INTERFACE I_XtsMover

PROPERTY Acceleration : mc_lreal
GET
END_GET
SET
END_SET
END_PROPERTY

METHOD ActivateTrack : HRESULT
VAR_INPUT
	Track : INT;
END_VAR
END_METHOD

METHOD ActivateZeroReferenceSystem : HRESULT
END_METHOD

PROPERTY ActualForce : LREAL
GET
END_GET
END_PROPERTY

PROPERTY ActualPosition : LREAL
GET
END_GET
END_PROPERTY

PROPERTY ActualTrackPosition : LREAL
GET
END_GET
END_PROPERTY

PROPERTY ActualVelocity : LREAL
GET
END_GET
END_PROPERTY

PROPERTY AxisRef : Reference to Axis_ref
GET
END_GET
END_PROPERTY

PROPERTY Deceleration : mc_lreal
GET
END_GET
SET
END_SET
END_PROPERTY

METHOD DisableMover : HRESULT
VAR_INPUT
END_VAR
END_METHOD

METHOD EnableMover : HRESULT
VAR_INPUT
END_VAR
END_METHOD

PROPERTY ErrorID : UDINT
GET
END_GET
END_PROPERTY

PROPERTY Gap : MC_LREAL
GET
END_GET
SET
END_SET
END_PROPERTY

METHOD GetActiveTrackLength : LREAL
VAR_INPUT
END_VAR
END_METHOD

METHOD GetMoverCtrlOTCID : XtsMoverControllerOTCID
VAR_INPUT
END_VAR
END_METHOD

METHOD HaltAxis : HRESULT
VAR_INPUT
END_VAR
END_METHOD

PROPERTY HasError : BOOL
GET
END_GET
END_PROPERTY

PROPERTY PUBLIC IdentInGroup : IDENT_IN_GROUP_REF
GET
END_GET
END_PROPERTY

PROPERTY IsActive : BOOL
GET
END_GET
END_PROPERTY

PROPERTY IsAMover1 : BOOL
GET
END_GET
END_PROPERTY

PROPERTY IsAvoidingCollision : BOOL
GET
END_GET
END_PROPERTY

PROPERTY IsDetected : BOOL
GET
END_GET
END_PROPERTY

PROPERTY IsEnabled : BOOL
GET
END_GET
END_PROPERTY

PROPERTY IsStationary : BOOL
GET
END_GET
END_PROPERTY

PROPERTY Jerk : mc_lreal
GET
END_GET
SET
END_SET
END_PROPERTY

PROPERTY PUBLIC MoversActiveTrack : INT
GET
END_GET
END_PROPERTY

PROPERTY PUBLIC MoverXtsIoEnvInterface : I_TcIoXtsXpuMover
GET
END_GET
SET
END_SET
END_PROPERTY

METHOD MoveTo : HRESULT
VAR_INPUT
	RequiredPosition : MC_LREAL;
	MoveVelocity : MC_LREAL;
	NonModuloMove : BOOL;
END_VAR
END_METHOD

PROPERTY MyCAGroup : I_CollisionGroup
GET
END_GET
SET
END_SET
END_PROPERTY

PROPERTY PositiveDirectionOnly : BOOL
GET
END_GET
SET
END_SET
END_PROPERTY

METHOD RegisterTracks : HRESULT
VAR_INPUT
	Track : I_XtsTrack;
END_VAR
END_METHOD

METHOD Reset : HRESULT
VAR_INPUT
END_VAR
END_METHOD

METHOD SetForceCouple : HRESULT
VAR_INPUT
	XtsMoverCtrlOTCID : Tc3_XTS_Utility.XtsMoverControllerOTCID;
END_VAR
END_METHOD

METHOD SetMoverActiveTrack : HRESULT
VAR_INPUT
	Track : INT;
END_VAR
END_METHOD

METHOD SetParameterSet : HRESULT
VAR_INPUT
	ParameterSet : OTCID;
END_VAR
END_METHOD

METHOD SetSimDetectionPartAndPosition : BOOL
VAR_INPUT
	Part : OTCID;
	Position : LREAL;
END_VAR
END_METHOD

METHOD TriggerMoverArrive : HRESULT
VAR_INPUT
END_VAR
END_METHOD

METHOD TriggerMoverLeave : HRESULT
VAR_INPUT
END_VAR
END_METHOD

END_INTERFACE

(* stored: Version 1.1.0.1
   Itf I_XtsMover: Id {3dcfc709-5ede-408c-bb46-9ff1ab7ba3a2}
   Folder Administration: Id {4954b02a-5467-474b-b4cc-9e953c27295d}
   Folder Commands: Id {106fb726-2896-4a76-8d42-ca08d03a1871}
   Folder Dynamics: Id {f06c35fd-2445-4fb9-97b8-caf92ac08b38}
   Folder Status: Id {6f079834-b92a-4de6-abe6-7b90d541a1af}
   Property Acceleration: Id {968dd06c-5bd7-474e-8a7d-3c6c7a848d78}
   Get Get: Id {ad3ccb1b-ebe0-4c79-851d-54fe9678941a}
   Set Set: Id {ad0cd55c-ffe5-41e5-89e5-44c936340625}
   Method ActivateTrack: Id {ba6e327e-25a9-4189-a1a0-64429eeca8b6}
   Method ActivateZeroReferenceSystem: Id {ab0eeb60-9673-46f5-be7f-8e50f8587ea1}
   Property ActualForce: Id {00e4b1c4-c6de-437f-8c1d-7314c009badc}
   Get Get: Id {ae9db5cd-10af-4e87-b4a2-e547ec5c553c}
   Property ActualPosition: Id {28cc63bc-e59d-4da9-a15c-a10a220bddfe}
   Get Get: Id {9cdf084e-f593-4336-8f01-56fe49195bb3}
   Property ActualTrackPosition: Id {e9f1d418-aa47-422b-9743-bf025f0e00db}
   Get Get: Id {5f8e75a9-0ebf-4529-928e-062c555b8cba}
   Property ActualVelocity: Id {4743bebc-3e65-4ae0-ae76-394e50299433}
   Get Get: Id {c9377cd8-6623-42ce-ab9c-71b02227228b}
   Property AxisRef: Id {b9459322-2642-4758-9d1a-f140abbed4b3}
   Get Get: Id {fca9e840-ce68-48f6-aaf7-b30da4df166b}
   Property Deceleration: Id {925224a3-633f-4afb-a6bb-5e2282bf0166}
   Get Get: Id {ee77943b-5dd1-4851-bfac-c1f6c08f427a}
   Set Set: Id {cf0b19b4-9657-4139-bc2e-afb49fbc4d88}
   Method DisableMover: Id {ab15092e-3fa3-489a-9dc6-5a5b357cf3f5}
   Method EnableMover: Id {12e4840c-ab85-431d-8aa9-ce712b4847e4}
   Property ErrorID: Id {b04c2e44-101b-40a1-bb51-ba2468016913}
   Get Get: Id {4e6c86e3-a90a-4b81-8f9a-ac29a4c9cc2b}
   Property Gap: Id {fb9a5121-dbab-42c7-b05b-e0e4367182c8}
   Get Get: Id {0b18224e-8e16-4474-96e3-0906bc0c9a81}
   Set Set: Id {2dea6ad0-842c-4a1e-91cb-fd845bae918b}
   Method GetActiveTrackLength: Id {5c2216e1-42a4-4136-9c70-0f82d23b2aef}
   Method GetMoverCtrlOTCID: Id {863e8ade-d7f2-439e-8b15-5f1837c580a0}
   Method HaltAxis: Id {881642ff-213b-4030-944f-bd624c008c64}
   Property HasError: Id {90e38746-64a9-412e-b69f-e80f2d788cc6}
   Get Get: Id {5d936f5b-33ae-4901-8b9f-50eb63a5b11c}
   Property IdentInGroup: Id {892b953d-abf1-49a8-bf89-421385c1791d}
   Get Get: Id {b023befb-8f40-468b-ada4-daaf368f7d24}
   Property IsActive: Id {43095e03-0781-4c14-aea8-4bb8d9b5c9a9}
   Get Get: Id {5c30f132-658c-45bd-986b-b41d82b1ab82}
   Property IsAMover1: Id {2bbcc45a-af5d-48fd-a64e-6509262e5e53}
   Get Get: Id {35cbc1b6-e96d-405e-9119-f59168018c94}
   Property IsAvoidingCollision: Id {5943782e-d40c-4ea0-9ddf-8fe8e953cf52}
   Get Get: Id {a0bd6fb0-24f5-415f-851e-6efe2481bd7c}
   Property IsDetected: Id {93c73707-2737-4a0d-b791-8a8c892ba285}
   Get Get: Id {5a7d46d0-a531-4a2d-8d8f-a2055343f49b}
   Property IsEnabled: Id {1dc642f1-9317-4da4-80d2-54b08fffd57c}
   Get Get: Id {0b3bdbce-a4ec-4a95-bc52-fef9dadad358}
   Property IsStationary: Id {08154e2f-b533-419e-9633-c8866a41fb11}
   Get Get: Id {4afa1b23-4ee3-47ce-9d91-4217690a4938}
   Property Jerk: Id {8063437d-ace9-4769-bdaf-bbbe2e6cdcb8}
   Get Get: Id {7a71a7bc-503a-407e-bd5c-807dc27f8a07}
   Set Set: Id {943274ff-ff90-4228-a079-22863adf0d58}
   Property MoversActiveTrack: Id {f033ba71-1699-4f66-8762-38178a524724}
   Get Get: Id {ab30b8a7-22d3-4a5c-a941-ce17b5400c54}
   Property MoverXtsIoEnvInterface: Id {192fc175-f0e7-4171-9425-47deb3799f9d}
   Get Get: Id {e7a8a250-ae9b-4ad7-bf97-7690d04cb985}
   Set Set: Id {f163ce07-1471-4036-baf2-4d783308d9bd}
   Method MoveTo: Id {ff1a94f0-d91e-4f1f-8540-ce9d25779d5e}
   Property MyCAGroup: Id {7bdbd73e-c8bd-4342-9139-b02fb8b34afa}
   Get Get: Id {02d1886c-e164-4472-af91-ae6725f23e23}
   Set Set: Id {0add7ecc-1e34-4c45-86ea-05d00a10668e}
   Property PositiveDirectionOnly: Id {ed0ab13d-fd6f-4b8b-a5b2-30d977b85665}
   Get Get: Id {ca7928e2-abd0-4257-bca9-4dcae3e4cfec}
   Set Set: Id {89d703fe-11d9-4067-a762-3ca15c65b604}
   Method RegisterTracks: Id {f708c3cc-b99d-4712-bcc3-26ae6f024fa0}
   Method Reset: Id {6858a2d4-c501-4639-b0f6-64db9416c8f9}
   Method SetForceCouple: Id {99e00719-7cb8-4a43-85db-8a5d5fa2d5af}
   Method SetMoverActiveTrack: Id {3fb3e9b5-fc2f-40d4-a659-03f62aab1916}
   Method SetParameterSet: Id {96f05e89-0ff7-461f-963a-bf5f28b369db}
   Method SetSimDetectionPartAndPosition: Id {b203fdbc-b34c-4c13-b77e-aae6fc3e86cf}
   Method TriggerMoverArrive: Id {ce200a85-cca0-47d0-8b7e-22e3d01f8c11}
   Method TriggerMoverLeave: Id {fe2ebe40-b0b7-4184-8656-d9f18bf6a0ec} *)
